TYPE ST_ZForceControlProfile : STRUCT
    (* Profile编号。 *)
    nProfileId : UDINT;
    (* Profile修订号；变化时必须执行积分无扰预置。 *)
    nRevision : UDINT;
    (* 速度前馈，向下为正，单位毫米每秒。 *)
    fVelocityFeedForwardMmS : LREAL;
    (* 比例增益，单位毫米每秒每千牛。 *)
    fKp : LREAL;
    (* 积分增益，单位毫米每二次方秒每千牛。 *)
    fKi : LREAL;
    (* 抗积分饱和回算增益，单位每秒。 *)
    fKaw : LREAL;
    (* 积分项绝对限幅，单位毫米每秒。 *)
    fIntegralLimit : LREAL;
    (* 向上最大速度，单位毫米每秒。 *)
    fMaxUpVelocityMmS : LREAL;
    (* 向下最大速度，单位毫米每秒。 *)
    fMaxDownVelocityMmS : LREAL;
    (* 最大加速度，单位毫米每二次方秒。 *)
    fMaxAccelerationMmS2 : LREAL;
    (* 制动距离裕量，单位毫米。 *)
    fBrakeMarginMm : LREAL;
    (* 设定力斜坡，单位牛顿每秒。 *)
    fForceRampNS : LREAL;
    (* 参数是否有效。 *)
    bValid : BOOL;
END_STRUCT
END_TYPE

(* stored: Version 1.1.0.1
   DUT ST_ZForceControlProfile: Id {D3100000-0000-4000-8000-000000000006} *)
